(* CODESYS project IceMakerSequence.xml

Project tree, tasks and I/O mapping:
  function block IceMakerSequence [SFC]
*)

// IceMakerSequence
FUNCTION_BLOCK IceMakerSequence
//  .					.					.
VAR_INPUT
	SFCInit: 			BOOL;
	NeedIce: 			BOOL;
	StirComplete: 		BOOL;
	MakeIceTimeout: 	TIME;
	FaultReset: 		BOOL;
END_VAR
VAR_OUTPUT
	StirIce: 			BOOL;
	MakeIce: 			BOOL;
	MakeIceFault: 		BOOL;
END_VAR
VAR
END_VAR

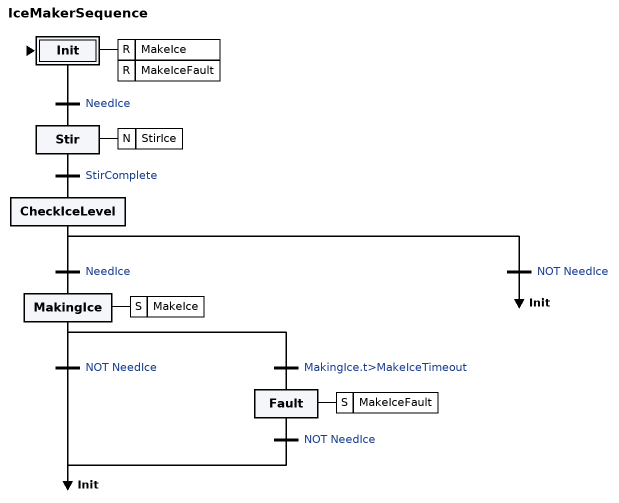
INITIAL_STEP Init:
    MakeIce(R);
    MakeIceFault(R);
END_STEP
TRANSITION FROM Init TO Stir
    := NeedIce;
END_TRANSITION
STEP Stir:
    StirIce(N);
END_STEP
TRANSITION FROM Stir TO CheckIceLevel
    := StirComplete;
END_TRANSITION
STEP CheckIceLevel:
END_STEP
TRANSITION FROM CheckIceLevel TO MakingIce
    := NeedIce;
END_TRANSITION
STEP MakingIce:
    MakeIce(S);
END_STEP
TRANSITION FROM MakingIce TO Init
    := NOT NeedIce;
END_TRANSITION
TRANSITION FROM MakingIce TO Fault
    := MakingIce.t>MakeIceTimeout;
END_TRANSITION
STEP Fault:
    MakeIceFault(S);
END_STEP
TRANSITION FROM Fault TO Init
    := NOT NeedIce;
END_TRANSITION
TRANSITION FROM CheckIceLevel TO Init
    := NOT NeedIce;
END_TRANSITION

END_FUNCTION_BLOCK
